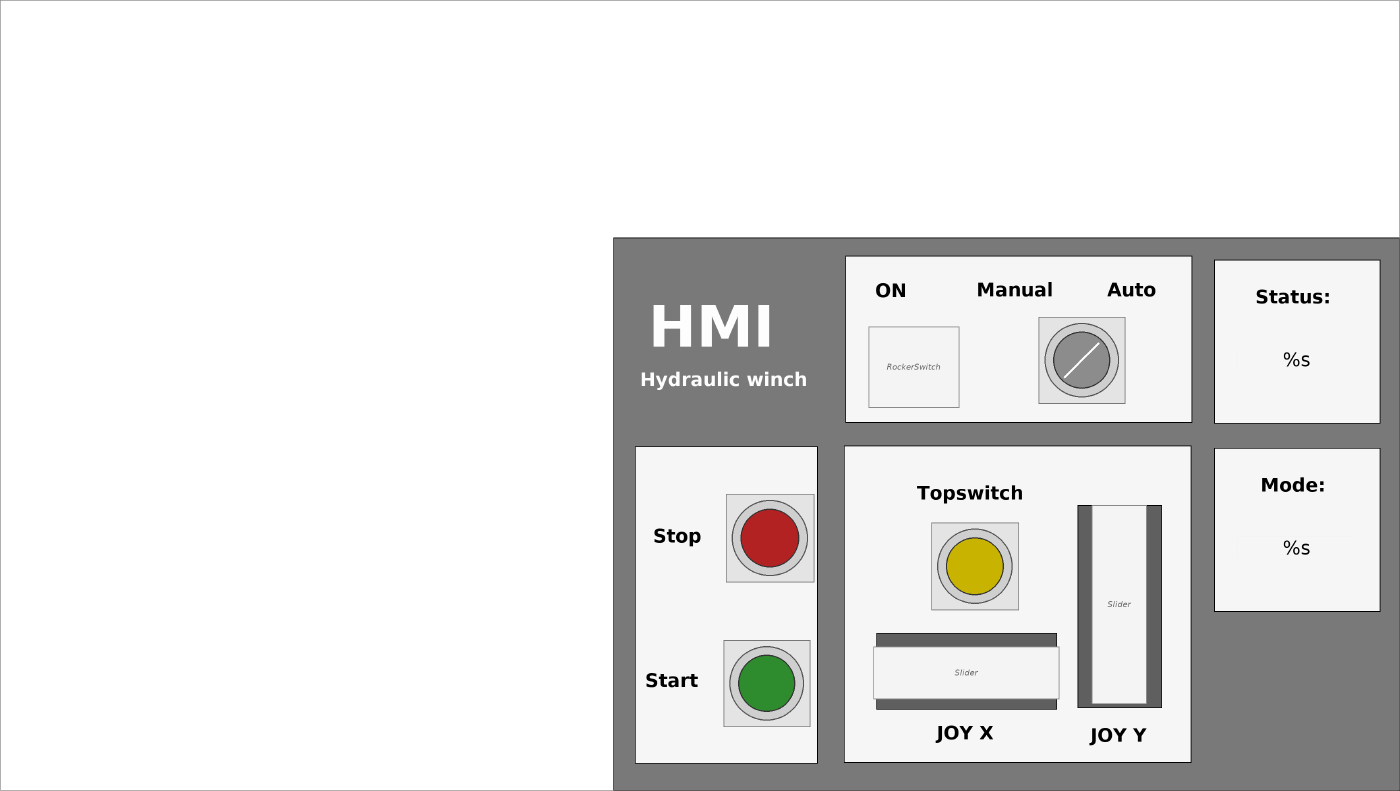
VISUALIZATION Visualization  // 1762x996
    Rectangle (772,299 990x697)
    RoundedRectangle (1528,327 209x206)
    RoundedRectangle (799,562 230x399)
    RoundedRectangle (1062,561 437x399)
    RoundedRectangle (1064,322 436x210)
    PushSwitch (899,622 140x111), variable: task1.bStop, behaviour: TAP, style: Switch-PushSwitch-Red
    PushSwitch (901,806 128x109), variable: task1.bStart, behaviour: TAP, style: Switch-PushSwitch-Green
    Label (774,815 143x84), "Start"
    Label (781,633 143x84), "Stop"
    RockerSwitch (1093,411 114x102), variable: task1.bOn, behaviour: TOGGLE, style: Switch-RockerSwitch-Gray
    RotarySwitch (1295,399 133x109), variable: task1.bManual, behaviour: TOGGLE, style: Switch-RotarySwitch-Gray
    PushSwitch (1171,658 112x110), variable: task1.bTopSwitch, behaviour: TOGGLE, style: Switch-PushSwitch-Yellow
    Label (1146,606 150x30), "Topswitch"
    Label (1333,909 150x34), "JOY Y"
    RoundedRectangle (1356,636 106x255)
    Slider (1374,636 69x250), variable: task1.fJoystickY, scale 11787..20509
    Label (1140,908 150x30), "JOY X"
    RoundedRectangle (1168,732 96x227), angle 270
    Slider (1099,814 234x66), variable: task1.fJoystickX, scale 11787..20509
    Label (1050,324 143x84), "ON"
    Label (1206,323 143x84), "Manual"
    Label (1353,323 143x84), "Auto"
    Label (792,367 232x88), "HMI"
    Label (795,434 232x88), "Hydraulic winch"
    Textfield (1557,438 150x30), "%s", text variable: task1.eStatus
    Label (1556,332 143x84), "Status:"
    RoundedRectangle (1528,564 209x206)
    Textfield (1557,675 150x30), "%s", text variable: task1.eModeSwitch
    Label (1556,569 143x84), "Mode:"
END_VISUALIZATION

(* stored: Version 1.1.0.1, ProductVersion 3.1.4024.12
   Visu Visualization: Id {7e46cb04-4e11-4884-a7f6-918fe33c6aed} *)
